FUNCTION_BLOCK TcoAiTests EXTENDS TcoCore._internals_TcoContext
VAR
	_signal : DINT;
	_sut : TcoElements.TcoAi(THIS^);
	_sutNotInitialized : TcoElements.TcoAi(THIS^);


END_VAR

VAR
	_ScaledResult: REAL;

END_VAR

METHOD PROTECTED Main
CASE _testId OF
    50:

        _sutNotInitialized.Service();
        _sutNotInitialized.Restore();
    100:
        _sut(inoSignal := _signal);

        _ScaledResult := _sut.Status.Scaled;

END_CASE
END_METHOD

END_FUNCTION_BLOCK

(* stored: Version 1.1.0.1, ProductVersion 3.1.4024.9
   POU TcoAiTests: Id {d06c66c5-2ff0-0b1f-0fa0-ba52007dc23b}, SpecialFunc None
   Method Main: Id {fb7a498b-b279-0615-3b52-7950031e3568} *)
